# EPICS substitutions: utcaApp/Db/fmcpico1m_4ch.substitutions
file db/fmcpico1m_4ch.template {
    pattern {ADDR}
	 {0}
	 {1}
	 {2}
	 {3}
}
